{attribute 'qualified_only'}
VAR_GLOBAL

(*
    Only includes motor definitions for the IOC
    These are hard-coded to be Main.M#,
    but are very convenient to store in a GVL,
    hence the confusing namespace here
    This should be refactored once the IOC
    supports arbitrary ads paths for motors
*)


    // Sample Chamber Sliding Seal - 1 axis
    //connect EPS limits
    {attribute 'pytmc' := 'pv: QRIX:SC:SSL:MMS'}
    {attribute 'TcLinkTo' := '.bLimitForwardEnable  := TIIB[EL7047_02_01 - SSL]^STM Status^Status^Digital input 1;
                              .bLimitBackwardEnable := TIIB[EL7047_02_01 - SSL]^STM Status^Status^Digital input 2;
                              .nRawEncoderULINT     := TIIB[EL5042_02_02]^FB Inputs Channel 1^Position'}
    M1: ST_MotionStage := (sName := 'QRIX:SSL:MMS');


    (* Start Adding Spectometer Arm Axes Here*)

    // 2Theta Stepper
    {attribute 'pytmc' := 'pv: QRIX:SA:MMS:2Theta'}
    {attribute 'TcLinkTo' := '	.bLimitForwardEnable  	:= TIIB[Rack#1A-04 DR_2Th (EL7047)]^STM Status^Status^Digital input 1;
                                .bLimitBackwardEnable 	:= TIIB[Rack#1A-04 DR_2Th (EL7047)]^STM Status^Status^Digital input 2;
                                .nRawEncoderULINT     	:= TIIB[Rack#1A-06 ENC_2Th (EL5042)]^FB Inputs Channel 1^Position;
                                .bBrakeRelease			:= TIIB[Rack#1A-05 MB_2Th (EL2602)]^Channel 1^Output
    '}
    M2: ST_MotionStage := (sName := 'QRIX:SA:MMS:2Theta');

    // XS1
    {attribute 'pytmc' := 'pv: QRIX:OPTSL:MMS:NORTH'}
    {attribute 'TcLinkTo' := '	.bLimitForwardEnable  	:= TIIB[Rack#2A-03 DR_XS1 (EL7041-0052)]^STM Status^Status^Digital input 1;
                                .bLimitBackwardEnable 	:= TIIB[Rack#2A-03 DR_XS1 (EL7041-0052)]^STM Status^Status^Digital input 2;
                                .nRawEncoderULINT     	:= TIIB[Rack#2B-07 ENC_X1_X2 (EL5042)]^FB Inputs Channel 1^Position
    '}
    M3: ST_MotionStage :=(sName := ' QRIX:OPTSL:MMS:NORTH');

    // XS2
    {attribute 'pytmc' := 'pv: QRIX:OPTSL:MMS:SOUTH'}
    {attribute 'TcLinkTo' := '	.bLimitForwardEnable  	:= TIIB[Rack#2A-04 DR_XS2 (EL7041-0052)]^STM Status^Status^Digital input 1;
                                .bLimitBackwardEnable 	:= TIIB[Rack#2A-04 DR_XS2 (EL7041-0052)]^STM Status^Status^Digital input 2;
                                .nRawEncoderULINT     	:= TIIB[Rack#2B-07 ENC_X1_X2 (EL5042)]^FB Inputs Channel 2^Position
    '}
    M4: ST_MotionStage:=(sName := ' QRIX:OPTSL:MMS:SOUTH');

    // YS1
    {attribute 'pytmc' := 'pv: QRIX:OPTSL:MMS:TOP'}
    {attribute 'TcLinkTo' := '	.bLimitForwardEnable  	:= TIIB[Rack#2A-05 DR_YS1 (EL7041-0052)]^STM Status^Status^Digital input 1;
                                .bLimitBackwardEnable 	:= TIIB[Rack#2A-05 DR_YS1 (EL7041-0052)]^STM Status^Status^Digital input 2;
                                .nRawEncoderULINT     	:= TIIB[Rack#2B-08 ENC_Y1_Y2 (EL5042)]^FB Inputs Channel 1^Position
    '}
    M5: ST_MotionStage:=(sName := ' QRIX:OPTSL:MMS:TOP');

    // YS2
    {attribute 'pytmc' := 'pv: QRIX:OPTSL:MMS:BOTTOM'}
    {attribute 'TcLinkTo' := '	.bLimitForwardEnable  	:= TIIB[Rack#2A-06 DR_YS2 (EL7041-0052)]^STM Status^Status^Digital input 1;
                                .bLimitBackwardEnable 	:= TIIB[Rack#2A-06 DR_YS2 (EL7041-0052)]^STM Status^Status^Digital input 2;
                                .nRawEncoderULINT     	:= TIIB[Rack#2B-08 ENC_Y1_Y2 (EL5042)]^FB Inputs Channel 1^Position
    '}
    M6: ST_MotionStage :=(sName := ' QRIX:OPTSL:MMS:BOTTOM');;

    // YG1
    {attribute 'pytmc' := 'pv: QRIX:OPT:MMS:Y1'}
    {attribute 'TcLinkTo' := '	.bLimitForwardEnable	:= TIIB[Rack#2A-10 DR_YG1 (EL7041-0052)]^STM Status^Status^Digital input 1;
                                .bLimitBackwardEnable	:= TIIB[Rack#2A-10 DR_YG1 (EL7041-0052)]^STM Status^Status^Digital input 2;
                                .nRawEncoderULINT		:= TIIB[Rack#2B-10 ENC_YG1_YG2 (EL5042)]^FB Inputs Channel 1^Position
    '}
    M7: ST_MotionStage:= (sName := 'QRIX:OPT:MMS:Y2');

    // YG2
    {attribute 'pytmc' := 'pv: QRIX:OPT:MMS:Y2'}
    {attribute 'TcLinkTo' := '	.bLimitForwardEnable	:= TIIB[Rack#2A-11 DR_YG2 (EL7041-0052)]^STM Status^Status^Digital input 1;
                                .bLimitBackwardEnable	:= TIIB[Rack#2A-11 DR_YG2 (EL7041-0052)]^STM Status^Status^Digital input 2;
                                .nRawEncoderULINT		:= TIIB[Rack#2B-10 ENC_YG1_YG2 (EL5042)]^FB Inputs Channel 2^Position
    '}
    M8: ST_MotionStage:= (sName := 'QRIX:OPT:MMS:Y2');

    // YG3
    {attribute 'pytmc' := 'pv: QRIX:OPT:MMS:Y3'}
    {attribute 'TcLinkTo' := '	.bLimitForwardEnable	:= TIIB[Rack#2A-12 DR_YG3 (EL7041-0052)]^STM Status^Status^Digital input 1;
                                .bLimitBackwardEnable	:= TIIB[Rack#2A-12 DR_YG3 (EL7041-0052)]^STM Status^Status^Digital input 2;
                                .nRawEncoderULINT		:= TIIB[Rack#2B-11 ENC_YG3_X1PM (EL5042)]^FB Inputs Channel 1^Position
    '}
    M9: ST_MotionStage:= (sName := 'QRIX:OPT:MMS:Y3');


    // RxG
    {attribute 'pytmc' := 'pv: QRIX:G:MMS:Rx'}
    {attribute 'TcLinkTo' := '	.bLimitForwardEnable	:= TIIB[Rack#2A-08 DR_RxG (EL7041-0052)]^STM Status^Status^Digital input 1;
                                .bLimitBackwardEnable	:= TIIB[Rack#2A-08 DR_RxG (EL7041-0052)]^STM Status^Status^Digital input 2;
                                .nRawEncoderULINT		:= TIIB[Rack#2B-09 ENC_RxG_XG (EL5042)]^FB Inputs Channel 1 compact^Position
    '}
    M10: ST_MotionStage:=(sName := 'QRIX:G:MMS:Rx');

    // XG
    {attribute 'pytmc' := 'pv: QRIX:G:MMS:X'}
    {attribute 'TcLinkTo' := '	.bLimitForwardEnable	:= TIIB[Rack#2A-09 DR_XG (EL7041-0052)]^STM Status^Status^Digital input 1;
                                .bLimitBackwardEnable	:= TIIB[Rack#2A-09 DR_XG (EL7041-0052)]^STM Status^Status^Digital input 2;
                                .nRawEncoderULINT		:= TIIB[Rack#2B-09 ENC_RxG_XG (EL5042)]^FB Inputs Channel 2^Position
    '}
    M11: ST_MotionStage:=(sName := 'QRIX:G:MMS:X');

    // XPM1
    {attribute 'pytmc' := 'pv: QRIX:PM:MMS:X1'}
    {attribute 'TcLinkTo' := '	.bLimitForwardEnable	:= TIIB[Rack#2A-14 DR_XPM1 (EL7041-0052)]^STM Status^Status^Digital input 1;
                                .bLimitBackwardEnable	:= TIIB[Rack#2A-14 DR_XPM1 (EL7041-0052)]^STM Status^Status^Digital input 2;
                                .nRawEncoderULINT		:= TIIB[Rack#2B-11 ENC_YG3_X1PM (EL5042)]^FB Inputs Channel 2^Position
    '}
    M12: ST_MotionStage :=(sName := 'QRIX:PM:MMS:X1');

    // XPM2
    {attribute 'pytmc' := 'pv: QRIX:PM:MMS:X2'}
    {attribute 'TcLinkTo' := '	.bLimitForwardEnable	:= TIIB[Rack#2A-15 DR_XPM2 (EL7041-0052)]^STM Status^Status^Digital input 1;
                                .bLimitBackwardEnable	:= TIIB[Rack#2A-15 DR_XPM2 (EL7041-0052)]^STM Status^Status^Digital input 2;
                                .nRawEncoderULINT		:= TIIB[Rack#2B-12 ENC_X2PM_RzPM (EL5042)]^FB Inputs Channel 1^Position
    '}
    M13: ST_MotionStage:=(sName := 'QRIX:PM:MMS:X2');

    // RzPM
    {attribute 'pytmc' := 'pv: QRIX:PM:MMS:Rz'}
    {attribute 'TcLinkTo' := '	.bLimitForwardEnable	:= TIIB[Rack#2A-16 DR_RzPM (EL7041-0052)]^STM Status^Status^Digital input 1;
                                .bLimitBackwardEnable	:= TIIB[Rack#2A-16 DR_RzPM (EL7041-0052)]^STM Status^Status^Digital input 2;
                                .nRawEncoderULINT		:= TIIB[Rack#2B-12 ENC_X2PM_RzPM (EL5042)]^FB Inputs Channel 2^Position
    '}
    M14: ST_MotionStage:=(sName := 'QRIX:PM:MMS:Rz');

    // YDF1
    {attribute 'pytmc' := 'pv: QRIX:DF:MMS:Y1'}
    {attribute 'TcLinkTo' := '	.bLimitForwardEnable  	:= TIIB[Rack#2B-15 DR_YDF1 (EL7041-0052)]^STM Status^Status^Digital input 1;
                                .bLimitBackwardEnable 	:= TIIB[Rack#2B-15 DR_YDF1 (EL7041-0052)]^STM Status^Status^Digital input 2
    '}
    M15: ST_MotionStage :=(sName := 'QRIX:DF:MMS:Y1');

    // YDF2
    {attribute 'pytmc' := 'pv: QRIX:DF:MMS:Y2'}
    {attribute 'TcLinkTo' := '	.bLimitForwardEnable  	:= TIIB[Rack#2B-16 DR_YDF2 (EL7041-0052)]^STM Status^Status^Digital input 1;
                                .bLimitBackwardEnable 	:= TIIB[Rack#2B-16 DR_YDF2 (EL7041-0052)]^STM Status^Status^Digital input 2
    '}
    M16: ST_MotionStage:=(sName := 'QRIX:DF:MMS:Y2');

    // YDF3
    {attribute 'pytmc' := 'pv: QRIX:DF:MMS:Y3'}
    {attribute 'TcLinkTo' := '	.bLimitForwardEnable  	:= TIIB[Rack#2B-19 DR_YDF3 (EL7041-0052)]^STM Status^Status^Digital input 1;
                                .bLimitBackwardEnable 	:= TIIB[Rack#2B-19 DR_YDF3 (EL7041-0052)]^STM Status^Status^Digital input 2
    '}
    M17: ST_MotionStage :=(sName := 'QRIX:DF:MMS:Y3');

    // XSDC1
    {attribute 'pytmc' := 'pv: QRIX:DETSL:MMS:NORTH'}
    {attribute 'TcLinkTo' := '	.bLimitForwardEnable  	:= TIIB[BOX-09 DR_XSDC1 (EL7041-0052)]^STM Status^Status^Digital input 1;
                                .bLimitBackwardEnable 	:= TIIB[BOX-09 DR_XSDC1 (EL7041-0052)]^STM Status^Status^Digital input 2;
                                .nRawEncoderULINT     	:= TIIB[BOX-03 ENC_X1_X2 (EL5042)]^FB Inputs Channel 1^Position
    '}
    M18: ST_MotionStage:=(sName := ' QRIX:DETSL:MMS:NORTH');

    // XSDC2
    {attribute 'pytmc' := 'pv: QRIX:DETSL:MMS:SOUTH'}
    {attribute 'TcLinkTo' := '	.bLimitForwardEnable	:= TIIB[BOX-10 DR_XSDC2 (EL7041-0052)]^STM Status^Status^Digital input 1;
                                .bLimitBackwardEnable 	:= TIIB[BOX-10 DR_XSDC2 (EL7041-0052)]^STM Status^Status^Digital input 2;
                                .nRawEncoderULINT     	:= TIIB[BOX-03 ENC_X1_X2 (EL5042)]^FB Inputs Channel 2^Position
    '}
    M19: ST_MotionStage :=(sName := ' QRIX:DETSL:MMS:SOUTH');

    // YSDC1
    {attribute 'pytmc' := 'pv: QRIX:DETSL:MMS:TOP'}
    {attribute 'TcLinkTo' := '	.bLimitForwardEnable	:= TIIB[BOX-11 DR_YSDC1 (EL7041-0052)]^STM Status^Status^Digital input 1;
                                .bLimitBackwardEnable 	:= TIIB[BOX-11 DR_YSDC1 (EL7041-0052)]^STM Status^Status^Digital input 2;
                                .nRawEncoderULINT     	:= TIIB[BOX-04 ENC_Y1_Y2 (EL5042)]^FB Inputs Channel 1^Position
    '}
    M20: ST_MotionStage :=(sName := ' QRIX:DETSL:MMS:TOP');

    // YSDC2
    {attribute 'pytmc' := 'pv: QRIX:DETSL:MMS:BOTTOM'}
    {attribute 'TcLinkTo' := '	.bLimitForwardEnable	:= TIIB[BOX-12 DR_YSDC2 (EL7041-0052)]^STM Status^Status^Digital input 1;
                                .bLimitBackwardEnable 	:= TIIB[BOX-12 DR_YSDC2 (EL7041-0052)]^STM Status^Status^Digital input 2;
                                .nRawEncoderULINT     	:= TIIB[BOX-04 ENC_Y1_Y2 (EL5042)]^FB Inputs Channel 1^Position
    '}
    M21: ST_MotionStage :=(sName := ' QRIX:DETSL:MMS:BOTTOM');

    // XDC
    {attribute 'pytmc' := 'pv: QRIX:DC:MMS:X'}
    {attribute 'TcLinkTo' := '	.bLimitForwardEnable  	:= TIIB[BOX-14 DR_XDC (EL7041-0052)]^STM Status^Status^Digital input 1;
                                .bLimitBackwardEnable 	:= TIIB[BOX-14 DR_XDC (EL7041-0052)]^STM Status^Status^Digital input 2;
                                .nRawEncoderULINT     	:= TIIB[BOX-05 ENC_XDC_RyDC (EL5042)]^FB Inputs Channel 1^Position
    '}
    M22: ST_MotionStage:=(sName := ' QRIX:DC:MMS:X');

    // RyDC
    {attribute 'pytmc' := 'pv: QRIX:DC:MMS:Ry'}
    {attribute 'TcLinkTo' := '	.bLimitForwardEnable	:= TIIB[BOX-15 DR_RyDC (EL7041-0052)]^STM Status^Status^Digital input 1;
                                .bLimitBackwardEnable	:= TIIB[BOX-15 DR_RyDC (EL7041-0052)]^STM Status^Status^Digital input 2;
                                .nRawEncoderULINT		:= TIIB[BOX-05 ENC_XDC_RyDC (EL5042)]^FB Inputs Channel 2^Position
    '}
    M23: ST_MotionStage :=(sName := ' QRIX:DC:MMS:Ry');

    // ZDC
    {attribute 'pytmc' := 'pv: QRIX:DC:MMS:Z'}
    {attribute 'TcLinkTo' := '	.bLimitForwardEnable	:= TIIB[BOX-16 DR_ZDC (EL7041-0052)]^STM Status^Status^Digital input 1;
                                .bLimitBackwardEnable	:= TIIB[BOX-16 DR_ZDC (EL7041-0052)]^STM Status^Status^Digital input 2;
                                .nRawEncoderULINT		:= TIIB[BOX-06 ENC_ZDC_YF1 (EL5042)]^FB Inputs Channel 1^Position
    '}
    M24: ST_MotionStage:=(sName := ' QRIX:DC:MMS:Z');

    // YF1
    {attribute 'pytmc' := 'pv: QRIX:DA:MMS:Y1'}
    {attribute 'TcLinkTo' := '	.bLimitForwardEnable	:= TIIB[Rack#1A-02 SFIN (EL1918)]^StandardInputs^Standard Out Var 10;
                                .bLimitBackwardEnable 	:= TIIB[Rack#1A-02 SFIN (EL1918)]^StandardInputs^Standard Out Var 11;
                                .nRawEncoderULINT     	:= TIIB[BOX-06 ENC_ZDC_YF1 (EL5042)]^FB Inputs Channel 2^Position;
                                .bBrakeRelease        	:= TIIB[BOX-19 MB_YF1_YF2 (EL2602)]^Channel 1^Output
    '}
    M25: ST_MotionStage:=(sName := ' QRIX:DA:MMS:Y1');

    // YF2
    {attribute 'pytmc' := 'pv: QRIX:DA:MMS:Y2'}
    {attribute 'TcLinkTo' := '	.bLimitForwardEnable	:= TIIB[Rack#1A-02 SFIN (EL1918)]^StandardInputs^Standard Out Var 12;
                                .bLimitBackwardEnable	:= TIIB[Rack#1A-02 SFIN (EL1918)]^StandardInputs^Standard Out Var 13;
                                .nRawEncoderULINT     	:= TIIB[BOX-07 ENC_YF2_ZF (EL5042)]^FB Inputs Channel 1^Position;
                                .bBrakeRelease			:= TIIB[BOX-19 MB_YF1_YF2 (EL2602)]^Channel 2^Output
    '}
    M26: ST_MotionStage:=(sName := ' QRIX:DA:MMS:Y2');

    // ZF
    {attribute 'pytmc' := 'pv: QRIX:DA:MMS:Z'}
    {attribute 'TcLinkTo' := '	.bLimitForwardEnable	:= TIIB[Rack#1A-02 SFIN (EL1918)]^StandardInputs^Standard Out Var 14;
                                .bLimitBackwardEnable	:= TIIB[Rack#1A-02 SFIN (EL1918)]^StandardInputs^Standard Out Var 15;
                                .nRawEncoderULINT		:= TIIB[BOX-07 ENC_YF2_ZF (EL5042)]^FB Inputs Channel 2^Position;
                                .bBrakeRelease			:= TIIB[Rack#2B-18 MB_ZF (EL2602)]^Channel 1^Output
    '}
    M27: ST_MotionStage:=(sName := ' QRIX:DA:MMS:Z');


    // Diffractometer -  8 axes START AT M28
    {attribute 'pytmc' := 'pv: QRIX:DIFF:MMS:X'}
    {attribute 'TcLinkTo' := '.bLimitForwardEnable  := TIIB[EL1088_03_04]^Channel 2^Input;
                              .bLimitBackwardEnable := TIIB[EL1088_03_04]^Channel 1^Input;
                              .bHome := TIIB[EL1088_03_10]^Channel 1^Input;
                              .nRawEncoderULINT     := TIIB[EL5042_03_02-Diff-X-Y]^FB Inputs Channel 1^Position'}
    M28: ST_MotionStage := (sName := 'QRIX:DIFF:MMS:X');

    {attribute 'pytmc' := 'pv: QRIX:DIFF:MMS:Y'}
    {attribute 'TcLinkTo' := '.bLimitForwardEnable  := TIIB[EL1088_03_04]^Channel 4^Input;
                              .bLimitBackwardEnable := TIIB[EL1088_03_04]^Channel 3^Input;
                              .bHome := TIIB[EL1088_03_10]^Channel 2^Input;
                              .nRawEncoderULINT     := TIIB[EL5042_03_02-Diff-X-Y]^FB Inputs Channel 2^Position'}
    M29: ST_MotionStage := (sName := 'QRIX:DIFF:MMS:Y');

    {attribute 'pytmc' := 'pv: QRIX:DIFF:MMS:Z'}
    {attribute 'TcLinkTo' := '.bLimitForwardEnable  := TIIB[EL1088_03_08]^Channel 2^Input;
                              .bLimitBackwardEnable := TIIB[EL1088_03_08]^Channel 1^Input;
                              .bHome := TIIB[EL1088_03_10]^Channel 3^Input;
                              .nRawEncoderULINT     := TIIB[EL5042_03_06-DIff-Z-2ThetaY]^FB Inputs Channel 1^Position'}
    M30: ST_MotionStage := (sName := 'QRIX:DIFF:MMS:Z');

    {attribute 'pytmc' := 'pv: QRIX:DIFF:MMS:DETY'}
    {attribute 'TcLinkTo' := '.bLimitForwardEnable  := TIIB[EL1088_03_08]^Channel 5^Input;
                              .bLimitBackwardEnable := TIIB[EL1088_03_08]^Channel 6^Input;
                              .bHome := TIIB[EL1088_03_10]^Channel 4^Input;
                              .nRawEncoderULINT     := TIIB[EL5042_03_06-DIff-Z-2ThetaY]^FB Inputs Channel 2^Position'}
    M31: ST_MotionStage := (sName := 'QRIX:DIFF:MMS:DETY');

    {attribute 'pytmc' := 'pv: QRIX:DIFF:MMS:PHI'}
    {attribute 'TcLinkTo' := '.bLimitForwardEnable  := TIIB[EL1088_03_08]^Channel 3^Input;
                              .bLimitBackwardEnable := TIIB[EL1088_03_08]^Channel 4^Input;
                              .bHome := TIIB[EL1088_03_10]^Channel 4^Input;
                              .nRawEncoderULINT     := TIIB[EL5042_03_13 - Diff - Phi - Chi]^FB Inputs Channel 1^Position'}
    M32: ST_MotionStage := (sName := 'QRIX:DIFF:MMS:PHI');

    {attribute 'pytmc' := 'pv: QRIX:DIFF:MMS:CHI'}
    {attribute 'TcLinkTo' := '.bLimitForwardEnable  := TIIB[EL1088_03_15]^Channel 2^Input;
                              .bLimitBackwardEnable := TIIB[EL1088_03_15]^Channel 1^Input;
                              .bHome := TIIB[EL1088_03_10]^Channel 6^Input;
                              .nRawEncoderULINT     := TIIB[EL5042_03_13 - Diff - Phi - Chi]^FB Inputs Channel 2^Position'}
    M33: ST_MotionStage := (sName := 'QRIX:DIFF:MMS:CHI');

    {attribute 'pytmc' := 'pv: QRIX:DIFF:MMS:THETA'}
    {attribute 'TcLinkTo' := '.bLimitForwardEnable  := TIIB[EL1088_03_15]^Channel 3^Input;
                              .bLimitBackwardEnable := TIIB[EL1088_03_15]^Channel 4^Input;
                              .bHome := TIIB[EL1088_03_10]^Channel 7^Input;
                              .nRawEncoderULINT     := TIIB[EL5042_03_17 - Diff - Theta - 2Theta]^FB Inputs Channel 1^Position'}
    M34: ST_MotionStage := (sName := 'QRIX:DIFF:MMS:THETA');

    {attribute 'pytmc' := 'pv: QRIX:DIFF:MMS:2THETA'}
    {attribute 'TcLinkTo' := '.bLimitForwardEnable  := TIIB[EL1088_03_15]^Channel 5^Input;
                              .bLimitBackwardEnable := TIIB[EL1088_03_15]^Channel 6^Input;
                              .bHome := TIIB[EL1088_03_10]^Channel 8^Input;
                              .nRawEncoderULINT     := TIIB[EL5042_03_17 - Diff - Theta - 2Theta]^FB Inputs Channel 2^Position'}
    M35: ST_MotionStage := (sName := 'QRIX:DIFF:MMS:2THETA');



    // Laser Table  -  3 axes
    {attribute 'pytmc' := 'pv: QRIX:LAS:MMS:VIS'}
    {attribute 'TcLinkTo' := '.bLimitForwardEnable  := TIIB[EL1088_02_06]^Channel 6^Input;
                              .bLimitBackwardEnable :=  TIIB[EL1088_02_06]^Channel 5^Input;
                              .nRawEncoderULINT     := TIIB[EL5042_02_05 - LAS_VIS]^FB Inputs Channel 1^Position'}
    M36: ST_MotionStage := (sName := 'QRIX:LAS:MMS:VIS');

    {attribute 'pytmc' := 'pv: QRIX:DIAG:MMS:H'}
    {attribute 'TcLinkTo' := '.bLimitForwardEnable  :=  TIIB[EL1088_02_06]^Channel 2^Input;
                              .bLimitBackwardEnable :=  TIIB[EL1088_02_06]^Channel 1^Input;
                              .nRawEncoderULINT     := TIIB[EL5042_02_08 - LAS_D_V-H]^FB Inputs Channel 2^Position'}
    M37: ST_MotionStage := (sName := 'QRIX:DIAG:MMS:H');

    {attribute 'pytmc' := 'pv: QRIX:DIAG:MMS:V'}
    {attribute 'TcLinkTo' := '.bLimitForwardEnable  := TIIB[EL1088_02_06]^Channel 4^Input;
                              .bLimitBackwardEnable := TIIB[EL1088_02_06]^Channel 3^Input;
                              .nRawEncoderULINT     := TIIB[EL5042_02_08 - LAS_D_V-H]^FB Inputs Channel 1^Position'}
    M38: ST_MotionStage := (sName := 'QRIX:DIAG:MMS:V');


    //Sample Delivery - 6 Axes


    {attribute 'pytmc' := 'pv: QRIX:SDS:MMS:X'}
    {attribute 'TcLinkTo' := '.bLimitForwardEnable  := TIIB[EL7047_04_01]^STM Status^Status^Digital input 1;
                              .bLimitBackwardEnable := TIIB[EL7047_04_01]^STM Status^Status^Digital input 2;
                              .nRawEncoderULINT     := TIIB[EL5042_04_02]^FB Inputs Channel 1^Position;
                              .bHome 				:= TIIB[EL1004_04_04]^Channel 1^Input'}
    M39: ST_MotionStage := (sName := 'QRIX:SDS:MMS:X');

    {attribute 'pytmc' := 'pv: QRIX:SDS:MMS:Y'}
    {attribute 'TcLinkTo' := '.bLimitForwardEnable  := TIIB[EL7047_04_03]^STM Status^Status^Digital input 2;
                              .bLimitBackwardEnable := TIIB[EL7047_04_03]^STM Status^Status^Digital input 1;
                              .nRawEncoderULINT     := TIIB[EL5042_04_02]^FB Inputs Channel 2^Position;
                              .bHome 				:= TIIB[EL1004_04_04]^Channel 2^Input'}
    M40: ST_MotionStage := (sName := 'QRIX:SDS:MMS:Y');

    {attribute 'pytmc' := 'pv: QRIX:SDS:MMS:Z'}
    {attribute 'TcLinkTo' := '.bLimitForwardEnable  := TIIB[EL7047_04_05]^STM Status^Status^Digital input 1;
                              .bLimitBackwardEnable := TIIB[EL7047_04_05]^STM Status^Status^Digital input 2;
                              .nRawEncoderULINT     := TIIB[EL5042_04_06]^FB Inputs Channel 1^Position;
                              .bHome 				:= TIIB[EL1004_04_04]^Channel 3^Input'}
    M41: ST_MotionStage := (sName := 'QRIX:SDS:MMS:Z');

     {attribute 'pytmc' := 'pv: QRIX:SDS:MMS:ROT_V'}
    {attribute 'TcLinkTo' := '.nRawEncoderUINT     := TIIB[EL5101_05_01]^ENC Status compact^Counter value;
                              .bHome 				:= TIIB[EL1004_04_04]^Channel 4^Input'}
    M42: ST_MotionStage := (sName := 'QRIX:SDS:MMS:ROT_V');

    {attribute 'pytmc' := 'pv: QRIX:SDS:MMS:ROT_H'}
    {attribute 'TcLinkTo' := '.bLimitForwardEnable  := TIIB[EL7047_04_10]^STM Status^Status^Digital input 2;
                              .bLimitBackwardEnable := TIIB[EL7047_04_10]^STM Status^Status^Digital input 1;
                              .nRawEncoderUINT     := TIIB[EL5101_05_02]^ENC Status compact^Counter value;
                              .bHome 				:= TIIB[EL1004_04_09]^Channel 1^Input'}
    M43: ST_MotionStage := (sName := 'QRIX:SDS:MMS:ROT_H');

    {attribute 'pytmc' := 'pv: QRIX:SDS:MMS:H'}
    {attribute 'TcLinkTo' := '.bLimitForwardEnable  := TIIB[EL7047_04_12]^STM Status^Status^Digital input 1;
                              .bLimitBackwardEnable := TIIB[EL7047_04_12]^STM Status^Status^Digital input 2;
                              .bHome 				:= TIIB[EL1004_04_09]^Channel 2^Input;
                              .nRawEncoderUINT     := TIIB[EL5101_05_03]^ENC Status compact^Counter value'}
    M44: ST_MotionStage := (sName := 'QRIX:SDS:MMS:H');

    //Detector Rotation
    {attribute 'pytmc' := 'pv: QRIX:DET:MMS:ROT'}
    {attribute 'TcLinkTo' := '.nRawEncoderULINT     := TIIB[BOX-22 DET_ROT (EL5042)]^FB Inputs Channel 1^Position'}
    M45: ST_MotionStage := (sName := 'QRIX:DET:MMS:ROT');

    // Cryo -  4 axes
    //Cryo -X
    {attribute 'pytmc' := 'pv: QRIX:CRYO:MMS:X'}
    {attribute 'TcLinkTo' := '.bLimitForwardEnable  := TIIB[EL7047_02_12]^STM Status^Status^Digital input 1;
                              .bLimitBackwardEnable := TIIB[EL7047_02_12]^STM Status^Status^Digital input 2;
                              .nRawEncoderULINT     := TIIB[EL5042_02_13]^FB Inputs Channel 1^Position'}
    M46: ST_MotionStage := (sName := 'QRIX:CRYO:MMS:X');
    //CRYO Y
    {attribute 'pytmc' := 'pv: QRIX:CRYO:MMS:Y'}
    {attribute 'TcLinkTo' := '.bLimitForwardEnable  := TIIB[EL7047_02_14]^STM Status^Status^Digital input 2;
                              .bLimitBackwardEnable := TIIB[EL7047_02_14]^STM Status^Status^Digital input 1;
                              .nRawEncoderULINT     := TIIB[EL5042_02_13]^FB Inputs Channel 2^Position'}
    M47: ST_MotionStage := (sName := 'QRIX:CRYO:MMS:Y');
    //CRYO Z
    {attribute 'pytmc' := 'pv: QRIX:CRYO:MMS:Z'}
    {attribute 'TcLinkTo' := '.bLimitForwardEnable  := TIIB[EL7047_02_15]^STM Status^Status^Digital input 1;
                              .bLimitBackwardEnable := TIIB[EL7047_02_15]^STM Status^Status^Digital input 2;
                              .nRawEncoderULINT     := TIIB[EL5042_02_16]^FB Inputs Channel 1^Position'}
    M48: ST_MotionStage := (sName := 'QRIX:CRYO:MMS:Z');
    // CRYO-ROT
    {attribute 'pytmc' := 'pv: QRIX:CRYO:MMS:ROT'}
    {attribute 'TcLinkTo' := '.bLimitForwardEnable  := TIIB[EL7047_02_11]^STM Status^Status^Digital input 1;
                              .bLimitBackwardEnable := TIIB[EL7047_02_11]^STM Status^Status^Digital input 2;
                              .nRawEncoderULINT     := TIIB[EL5042_02_16]^FB Inputs Channel 2^Position'}
    M49: ST_MotionStage := (sName := 'QRIX:CRYO:MMS:ROT');

(*
    // Questar -  2 axes
    {attribute 'pytmc' := 'pv: QRIX:QUESTAR:MMS:01'}
    {attribute 'TcLinkTo' := '.bLimitForwardEnable  := TIIB[SSL-EL7041]^STM Status^Status^Digital input 1;
                              .bLimitBackwardEnable := TIIB[SSL-EL7041]^STM Status^Status^Digital input 2;
                              .nRawEncoderULINT     := TIIB[IM1K3-EL5042]^FB Inputs Channel 1^Position'}
    M49: ST_MotionStage := (sName := 'QRIX:QUESTAR:MMS:01');

    {attribute 'pytmc' := 'pv: QRIX:QUESTAR:MMS:02'}
    {attribute 'TcLinkTo' := '.bLimitForwardEnable  := TIIB[SSL-EL7041]^STM Status^Status^Digital input 1;
                              .bLimitBackwardEnable := TIIB[SSL-EL7041]^STM Status^Status^Digital input 2;
                              .nRawEncoderULINT     := TIIB[IM1K3-EL5042]^FB Inputs Channel 1^Position'}
    M50: ST_MotionStage := (sName := 'QRIX:QUESTAR:MMS:02');
*)

END_VAR

(* stored: Version 1.1.0.1, ProductVersion 3.1.4022.18
   GVL Main: Id {2b6c7284-966c-4508-b749-c66dc5cfc539} *)
